INTERFACE I_AnalogInput

END_INTERFACE

(* stored: Version 1.1.0.1, ProductVersion 3.1.4026.18
   Itf I_AnalogInput: Id {13465ec1-a24c-49f9-b252-c5023320b0c4} *)
